// TIA Portal V16 export
// export: Created 2022-11-17T15:49:41.3112394Z, ExportSetting WithDefaults, DisplayName Totally Integrated Automation Portal, DisplayVersion V16 Update 6, DisplayName TIA Portal Version Control Interface, DisplayVersion V16 Update 2, DisplayName TIA Portal Openness, DisplayVersion V16 Update 6, DisplayName SINAMICS Startdrive Advanced, DisplayVersion V16 Update 5, DisplayName SINAMICS Startdrive G130, G150, S120, S150, SINAMICS MV, S210, DisplayVersion V16 Update 5, DisplayName SINAMICS Startdrive G110M, G120, G120C, G120D, G120P, G115D, DisplayVersion V16 Update 5, DisplayName STEP 7 Professional, DisplayVersion V16 Update 6, DisplayName STEP 7 Safety, DisplayVersion V16, DisplayName WinCC Advanced, DisplayVersion V16 Update 6
DATA_BLOCK "DB91_NetDB"   // DB91
{ S7_Optimized_Access := 'FALSE' }
VERSION : 0.1
// stored: AutoNumber false, IsOnlyStoredInLoadMemory false, IsWriteProtectedInAS false
   VAR RETAIN
      In_livebit : Bool := FALSE;   // set this bit to TRUE
      spare1 : Bool := FALSE;
      spare2 : Bool := FALSE;
      spare3 : Bool := FALSE;
      spare4 : Bool := FALSE;
      spare5 : Bool := FALSE;
      spare6 : Bool := FALSE;
      spare7 : Bool := FALSE;
      IN_PRI : Bool := FALSE;   // Pallet ready in infeed
      IN_RRO : Bool := FALSE;   // Ready to receive in outfeed
      IN_ETO : Bool := FALSE;   // End of transfer in outfeed
      IN_EXC : Bool := FALSE;   // Wrapping excluded signal
      IN_ResetPartial : Bool := FALSE;   // Reset partial wrapped counter
      IN_spare5 : Bool := FALSE;
      IN_spare6 : Bool := FALSE;
      IN_spare7 : Bool := FALSE;
      IN_Program : Byte := 16#00;   // Program selection byte 1-15 (0 excluded)
      OUT_RRI : Bool := FALSE;   // Ready to receive in infeed signal
      OUT_ETI : Bool := FALSE;   // End of transfer in infeed signal
      OUT_PRO : Bool := FALSE;   // Pallet ready in outfeed signal
      OUT_spare3 : Bool := FALSE;
      OUT_spare4 : Bool := FALSE;
      OUT_spare5 : Bool := FALSE;
      OUT_spare6 : Bool := FALSE;
      Out_LiveBit : Bool := FALSE;   // This bit always TRUE
      spare_word : Word := 16#0000;
      MachineStatus : Word := 16#0000;
      WorkedHours : DWord := 16#0000_0000;
      PalletWrapped : DWord := 16#0000_0000;
      PartialWrapped : DWord := 16#0000_0000;
      VD2300 : DWord := 16#0000_0000;
      VD2304 : DWord := 16#0000_0000;
      VD2308 : DWord := 16#0000_0000;
      VD2312 : DWord := 16#0000_0000;
      VD2316 : DWord := 16#0000_0000;
      VD2320 : DWord := 16#0000_0000;
      VD2324 : DWord := 16#0000_0000;
      VW2328 : Word := 16#0000;
   END_VAR
BEGIN
END_DATA_BLOCK
